FUNCTION_BLOCK TIMESERIES_CORRELATION_ANALYSIS
  {SET_ATTRIBUTE(OpcUa, SERVICE)}
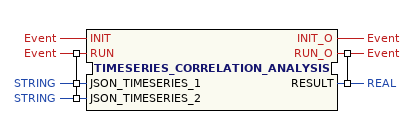
  EVENT_INPUT
    INIT;
    RUN WITH JSON_TIMESERIES_1, JSON_TIMESERIES_2;
  END_EVENT
  EVENT_OUTPUT
    INIT_O;
    RUN_O WITH RESULT;
  END_EVENT
  VAR_INPUT
    JSON_TIMESERIES_1 : STRING; {SET_ATTRIBUTE(OpcUa, Variable.RUN)}
    JSON_TIMESERIES_2 : STRING; {SET_ATTRIBUTE(OpcUa, Variable.RUN)}
  END_VAR
  VAR_OUTPUT
    RESULT : REAL; {SET_ATTRIBUTE(OpcUa, Variable.RUN)}
  END_VAR
END_FUNCTION_BLOCK
